// TIA Portal V17 export
// export: Created 2023-02-22T16:41:02.5134246Z, ExportSetting WithDefaults, DisplayName Totally Integrated Automation Portal, DisplayVersion V17, DisplayName TIA Portal Openness, DisplayVersion V17, DisplayName TIA Portal Version Control Interface, DisplayVersion V17, DisplayName TIA Portal Test Suite Advanced, DisplayVersion V17, DisplayName STEP 7 Professional, DisplayVersion V17, DisplayName SIMATIC Energy Suite, DisplayVersion V17, DisplayName STEP 7 Safety, DisplayVersion V17, DisplayName WinCC Professional, DisplayVersion V17
VAR_GLOBAL   // PLC tag table "Input"
   I_D1 AT %I0.0 : Bool;
   I_D2 AT %I0.1 : Bool;
   I_D3 AT %I0.2 : Bool;
   I_D4 AT %I0.3 : Bool;
   I_D5 AT %I0.4 : Bool;
   I_D6 AT %I0.5 : Bool;
   I_D7 AT %I0.6 : Bool;
   I_D8 AT %I0.7 : Bool;
   I_D9 AT %I1.0 : Bool;
   I_Start AT %I1.1 : Bool;
   I_Reset AT %I1.2 : Bool;
   I_Stop AT %I1.3 : Bool;
   I_Auto AT %I1.4 : Bool;
   I_Manual AT %I1.5 : Bool;
   I_Estop AT %I1.6 : Bool;
   I_C1 AT %I1.7 : Bool;
   I_C2 AT %I2.0 : Bool;
   I_C3 AT %I2.1 : Bool;
   I_C4 AT %I2.2 : Bool;
   I_C5 AT %I2.3 : Bool;
   I_SendLeft AT %I2.4 : Bool;
   I_SendForward AT %I2.5 : Bool;
   I_SendRight AT %I2.6 : Bool;
   I_ResetCount AT %I2.7 : Bool;
   I_Weight AT %ID30 : Real;
END_VAR
